//IP v4 address as an union to provide the address in a UDINT and array format 
TYPE U_IPv4Addr : 
UNION
	Stacked 				: UDINT; //IPv4 address combined in a UDINT
	Bytes 					: T_IPv4AddrArr; //IPv4 address as an array 0..3 of Byte
END_UNION
END_TYPE

(* stored: Version 1.1.0.1, ProductVersion 3.1.4022.3
   DUT U_IPv4Addr: Id {74f50984-7cee-4d59-acb7-443e0a659645} *)
